FUNCTION_BLOCK "CM_DRVT_N"   // FB148, SCL
{ S7_Optimized_Access := 'FALSE' }
VERSION : 0.0
// --------------------------------------------------------------------------------
//     program     :    CM_DRVT_N
//     description :    calculation of derivative to the order n 
//     name        :    G. Eibelsh鋟ser
//     date        :    31.01.2007
// 
//     revision    :  
//     name        :   
//     date        :    
// 
//                     (c)CGS
//     --------------------------------------------------------------------------------
   VAR_INPUT
      calc_on : Bool;   // calculation activated
      order : Int;   // order of first derivation
      u_in : Real;   // input value
      ts_in : Real;   // sample time
      tc_in : Real;   // call time
      tme_base : Real;
   END_VAR
   VAR_IN_OUT
      y_out : Real;   // output value
   END_VAR
   VAR
      data_rec_init : Bool;   // data record initialisation
      calc_cycle : Int;   // calculation cycle
      i : Int;   // record index
      t : Int;   // time between newest and oldest value in record
      y_t : Real;   // newest value in data record
      y_tn : Real;   // oldest value in data record
      data_rec : Array[0..3600] of Real;   // data record
   END_VAR
BEGIN


       IF #calc_on  THEN        //caculation enabled
           IF #calc_cycle >= REAL_TO_INT(#ts_in / #tc_in)   THEN 
               #calc_cycle  :=  1;

               IF (#order > 3600)   THEN
                   #order   :=  3600;       //limit order to a maximum of 3600
               END_IF;

               IF (#order > 0)  THEN //order of first derivation must be >0

                   //read oldest value from data record
                   //----------------------------------
                   IF (#i = 0) AND #data_rec_init THEN   //record initialisation with new values 
                       #y_tn    :=  #u_in;               //keep y_tn on first input during initialisation
                   ELSIF NOT #data_rec_init THEN 
                       #y_tn    :=  #data_rec[#i];        //write oldest record data to y_tn before overwritting it
                   END_IF;

                   //store new input value in record
                   //-------------------------------
                   #data_rec[#i] :=  #u_in;

                   //read newest value from data record
                   //----------------------------------
                   #y_t :=  #data_rec[#i];

                   //calculation of time between newest and oldest value in record
                   //-------------------------------------------------------------
                   IF #data_rec_init    THEN
                       #t   :=  #i;
                   ELSE
                       #t   :=  #order;
                   END_IF;

                   //calculate first derivation and scale
                   //------------------------------------
                   IF (#t > 0) THEN 
                       #y_out   :=  ((#y_t - #y_tn) / #t) * (#tme_base / #ts_in);
                   END_IF;

                   //increment record index each call
                   //--------------------------------
                   #i   :=  #i + 1;

                   //reset record index when maximum amount of values is reached
                   //-----------------------------------------------------------
                   IF (#i > #order)  THEN
                       #i               :=  0;
                       #data_rec_init   :=  FALSE;
                   END_IF;
               END_IF;
           ELSE   
               #calc_cycle  :=  #calc_cycle + 1;
           END_IF;

       //caculation disabled - reset variables and flags
       //-----------------------------------------------
       ELSE                
           #i               :=  0;
           #y_out           :=  0.0;
           #calc_cycle      :=  1;
           #data_rec_init   :=  TRUE;

       END_IF;
END_FUNCTION_BLOCK

FUNCTION_BLOCK "CM_CALC"   // FB149, SCL
{ S7_Optimized_Access := 'FALSE' }
VERSION : 0.0
// --------------------------------------------------------------------------------
//     program     :    CM_CALC
//     description :    filter calculations 
//     name        :    G. Eibelsh鋟ser
//     date        :    01.07.2020 
// 
//     revision    :    
//     name        :    
//     date        :    
// 
//                     (c)PVA TePla AG
//     --------------------------------------------------------------------------------
   VAR
      S_CAM_1_CTR_X : "CM_PT1";   // PT1
      S_CAM_2_CTR_X : "CM_PT1";   // PT1
      S_CAM_1_RAD_PT : "CM_PT1";   // PT1
      S_CAM_2_RAD_PT : "CM_PT1";   // PT1
      S_CAM_1_DIA_CF : "CM_PT2";   // PT2
      S_CAM_2_DIA_CF : "CM_PT2";   // PT2
      S_CAM_XT_DIA : "CM_PT2";   // PT2
      S_CAM_MLT_LVL_CHG : "CM_PT1";   // PT1
      i : Int;
      scam_mlt_lvl_t1 : Real;
   END_VAR
   VAR CONSTANT
      x_resolution : Real := 2063.0;
      mlt_lvl_chg_rng : Real := 100.0;
   END_VAR
BEGIN

       //stereo camera
       //-------------
       //center x- coordinate of circle fit camera 1
       //-------------------------------------------
       #S_CAM_1_CTR_X  (u_in      := "AV".S_CAM_1_ACT_CF_CTR_X,   //read actual pixel value                  
                       t1_in     := 15.0,                      //delay time T1
                       ts_in     := 0.1,
                       tc_in     := 0.1,
                       range_in  := #x_resolution,
                       range_out := #x_resolution,
                       y_llim    := 0.0,
                       y_hlim    := #x_resolution,
                       y_out     := "AV".S_CAM_1_AVG_CF_CTR_X);  //write average value - not used

       //center x- coordinate of circle fit camera 2
       //-------------------------------------------
       #S_CAM_2_CTR_X  (u_in      := "AV".S_CAM_2_ACT_CF_CTR_X,   //read actual pixel value                    
                       t1_in     := 15.0,                      //delay time T1
                       ts_in     := 0.1,
                       tc_in     := 0.1,
                       range_in  := #x_resolution,
                       range_out := #x_resolution,
                       y_llim    := 0.0,
                       y_hlim    := #x_resolution,
                       y_out     := "AV".S_CAM_2_AVG_CF_CTR_X);  //write average value - not used

       //radius point of camera 1
       //------------------------
       #S_CAM_1_RAD_PT (u_in      := "AV".S_CAM_1_ACT_RAD_PT,     //read actual pixel value                  
                       t1_in     := 15.0,                      //delay time T1
                       ts_in     := 0.1,
                       tc_in     := 0.1,
                       range_in  := #x_resolution,
                       range_out := #x_resolution,
                       y_llim    := 0.0,
                       y_hlim    := #x_resolution,
                       y_out     := "AV".S_CAM_1_AVG_RAD_PT);    //write average value - used for calculation of delta_r and delta_h

       //radius point of camera 2
       //------------------------
       #S_CAM_2_RAD_PT (u_in      := "AV".S_CAM_2_ACT_RAD_PT,     //read actual pixel value                  
                       t1_in     := 15.0,                      //delay time T1
                       ts_in     := 0.1,
                       tc_in     := 0.1,
                       range_in  := #x_resolution,
                       range_out := #x_resolution,
                       y_llim    := 0.0,
                       y_hlim    := #x_resolution,
                       y_out     := "AV".S_CAM_2_AVG_RAD_PT);    //write average value - used for calculation of delta_r and delta_h

       //circle fit camera 1 - PT 2 call
       //-------------------------------
       #S_CAM_1_DIA_CF (u_in      := "AV".S_CAM_1_ACT_DIA_CF,     //read actual pixel value                  
                       t1_in     := "AC".CTL_DIA_TF_1,           //delay time T1 - recipe parameter
                       t2_in     := "AC".CTL_DIA_TF_2,           //delay time T2 - recipe parameter
                       ts_in     := 0.1,
                       tc_in     := 0.1,
                       range_in  := #x_resolution,
                       range_out := #x_resolution,
                       y_llim    := 0.0,
                       y_hlim    := #x_resolution,
                       y_out     := "AV".S_CAM_1_AVG_DIA_CF);    //write average value - not used

       //circle fit camera 2 - PT 2 call
       //-------------------------------
       #S_CAM_2_DIA_CF (u_in      := "AV".S_CAM_2_ACT_DIA_CF,     //read actual pixel value                  
                       t1_in     := "AC".CTL_DIA_TF_1,           //delay time T1 - recipe parameter
                       t2_in     := "AC".CTL_DIA_TF_2,           //delay time T2 - recipe parameter
                       ts_in     := 0.1,
                       tc_in     := 0.1,
                       range_in  := #x_resolution,
                       range_out := #x_resolution,
                       y_llim    := 0.0,
                       y_hlim    := #x_resolution,
                       y_out     := "AV".S_CAM_2_AVG_DIA_CF);    //write average value - not used

       //actual crystal diameter - PT 2 call
       //-----------------------------------
       #S_CAM_XT_DIA   (u_in      := "AV".S_CAM_ACT_XT_DIA,       //read actual mm value                  
                       t1_in     := "AC".CTL_DIA_TF_1,           //delay time T1 - recipe parameter
                       t2_in     := "AC".CTL_DIA_TF_2,           //delay time T2 - recipe parameter
                       ts_in     := 0.1,
                       tc_in     := 0.1,
                       range_in  := "CNF".XT_DIA_RANGE,
                       range_out := "CNF".XT_DIA_RANGE,
                       y_llim    := 0.0,
                       y_hlim    := "CNF".XT_DIA_RANGE,
                       y_out     := "AV".S_CAM_AVG_XT_DIA);      //write average value - used for control loop

       //reset filter time to zero while melt level variable is reseted
       //--------------------------------------------------------------
       IF ("LT".RST_MLT_LVL AND (#i <= 5)) THEN
           #scam_mlt_lvl_t1     :=  0.0;
           #i                   :=  #i + 1;
       ELSE
           #scam_mlt_lvl_t1     :=  "PAR_SUB".SCAM_MLT_LVL_T1;
           "LT".RST_MLT_LVL      :=  FALSE;
           #i                   :=  0;
       END_IF;

       //actual crystal melt level change
       //--------------------------------
       #S_CAM_MLT_LVL_CHG  (u_in      := "AV".S_CAM_ACT_MLT_LVL_CHG,      //read actual mm value                  
                           t1_in     := #scam_mlt_lvl_t1,               //delay time T1
                           ts_in     := 0.1,
                           tc_in     := 0.1,
                           range_in  := #mlt_lvl_chg_rng,
                           range_out := #mlt_lvl_chg_rng,
                           y_llim    := #mlt_lvl_chg_rng * (-1),
                           y_hlim    := #mlt_lvl_chg_rng,
                           y_out     := "AV".S_CAM_AVG_MLT_LVL_CHG);     //write average value - used for control loop

       //write display values
       //--------------------                 
       "DIS".S_CAM_ACT_XT_DIA        :=  "AV".S_CAM_AVG_XT_DIA;     
       "DIS".S_CAM_ACT_MLT_LVL_CHG   :=  "AV".S_CAM_AVG_MLT_LVL_CHG;
       "DIS".S_CAM_1_ACT_RAD_PT      :=  "AV".S_CAM_1_AVG_RAD_PT;
       "DIS".S_CAM_2_ACT_RAD_PT      :=  "AV".S_CAM_2_AVG_RAD_PT;
END_FUNCTION_BLOCK

FUNCTION_BLOCK "CM_DIA_CALC"   // FB150, SCL
{ S7_Optimized_Access := 'FALSE' }
VERSION : 0.0
// --------------------------------------------------------------------------------
//     program     :    CM_DIA_CALC
//     description :    calculation of crystal diameter from measured weight signal 
//     name        :    G. Eibelsh鋟ser
//     date        :    12.02.2008
// 
//                     diameter = 2 * SQRT(weight rate / (position increment * PI * density)
// 
//     revision    :  
//     name        :   
//     date        :    
// 
//                     (c)CGS
//     --------------------------------------------------------------------------------
   VAR_INPUT
      calc_on : Bool;   // calculation activated
      ts_in : Real;   // sample time
      tc_in : Real;   // call time
      u_in : Real;   // input value
      pos_inc : Real;
      pi : Real;
      rho_si_sol : Real;
   END_VAR
   VAR_IN_OUT
      y_out : Real;   // output value
   END_VAR
   VAR
      calc_cycle : Int;   // calculation cycle
   END_VAR
BEGIN


       IF #calc_on  THEN        //caculation enabled
           //do calculation
           //--------------
           IF #calc_cycle >= REAL_TO_INT(#ts_in / #tc_in)   THEN  //check calculation cycle 
               #calc_cycle  :=  1;
               //calculate diameter in mm
               //------------------------
               IF (#u_in > 0.0) AND (#pos_inc > 0.0) THEN 
                   #y_out   :=  2 * SQRT(#u_in / (#pos_inc * #pi * #rho_si_sol));          
               END_IF;
           ELSE   
               #calc_cycle  :=  #calc_cycle + 1; //increment calc cycle variable
           END_IF;

       //caculation disabled - reset output variable
       //-------------------------------------------
       ELSE                
           #calc_cycle      :=  1;
           #y_out           :=  0.0;

       END_IF;
END_FUNCTION_BLOCK

FUNCTION_BLOCK "CM_LOOP_AVG_GAP_OFFS"   // FB151, SCL
{ S7_Optimized_Access := 'FALSE' }
VERSION : 0.0
// --------------------------------------------------------------------------------
//     program     :    CM_LOOP_AVG_GAP_OFFS
//     description :    average gap offset controller
//     name        :    G. Eibelsh鋟ser
//     date        :    27.08.2020
// 
//     revision    :    
//     name        :    
//     date        :    
// 
//                     (c)PVA TePla AG
//     --------------------------------------------------------------------------------
   VAR
      GAP_OFFS : "CM_PT1";   // pt1 filter for average offset speed
      AVG_GAP_OFFS : CONT_C;   // Controller for offset speed of the gap control
      int_hold_req : Bool;   // integral hold action request
      ctrl_calls : Int;   // controller call counter
   END_VAR
   VAR_TEMP
      high_lim_active : Bool;   // high limit of controller output is reached
      low_lim_active : Bool;   // low limit of controller output is reached
      int_action_on : Bool;   // integral action on
      der_action_on : Bool;   // derivative action on
      per_out : Word;   // peripherial controller output variable
      p_part_out : Real;   // proportionality component
      i_part_out : Real;   // integral component
      d_part_out : Real;   // derivative component
      eff_act_val : Real;   // effective process variable
      error_sig : Real;   // control deviation
   END_VAR
   VAR CONSTANT
      nc : Real := 0.0;   // "not connected" input
   END_VAR
BEGIN

       //switch on average gap offset control
       //------------------------------------
       IF ("APC".AUTOMATIC AND "SY".CTL_OFFS_SPEED_ON AND NOT "SY".CTL_HTR_1_SMI) THEN        //offset speed control is triggered by gap control on
           "SY".CTL_AVG_OFFS_ON  :=  TRUE;
       ELSE
           "SY".CTL_AVG_OFFS_ON  :=  FALSE;
       END_IF;    

       //call filter algorithm
       //---------------------                                                  
       #GAP_OFFS(u_in       := "CTL".SET_GAP_CTL_OFFS,                          
               t1_in       := "PAR_MAIN".CTL_AVG_GAP_OFFS_TF, 
               ts_in       := 0.1,
               tc_in       := 0.1,
               range_in    := "CNF".MAX_GAP_OFFS,
               range_out   := "CNF".MAX_GAP_OFFS,
               y_llim      := "CNF".MAX_GAP_OFFS * (-1.0),
               y_hlim      := "CNF".MAX_GAP_OFFS,
               y_out       := "CTL".AVG_GAP_CTL_OFFS); 

       //enable of single controller actions
       //----------------------------------- 
       IF ("AC".CTL_AV_OFFS_TI > 0.0)   THEN         //i- part
           #int_action_on   :=  true;
       ELSE
           #int_action_on   :=  false;
       END_IF;

       IF ("AC".CTL_AV_OFFS_TD > 0.0)   THEN         //d-part
           #der_action_on   :=  true;
       ELSE
           #der_action_on   :=  false;
       END_IF;

       //call average gap offset controller 
       //----------------------------------
       #AVG_GAP_OFFS(COM_RST        :=  "KYD".OFFS_CTRL_RST,                  //restart of controller, resets controller values
                   MAN_ON          :=  NOT "SY".CTL_AVG_OFFS_ON,             //switch controller on/off
                   PVPER_ON        :=  false,                              //activate reading of peripherie value
                   P_SEL           :=  true,                               //proportional action on
                   I_SEL           :=  #int_action_on,                      //integral action on
                   INT_HOLD        :=  #int_hold_req,                       //integral action hold
                   I_ITL_ON        :=  false,                              //initialization of the integral action - set value of I_ITLVAL
                   D_SEL           :=  #der_action_on,                      //derivative action on
                   CYCLE           :=  T#100ms,                            //sample time
                   SP_INT          :=  0.0,                                //internal setpoint
                   PV_IN           :=  "CTL".AVG_GAP_CTL_OFFS * (-1),        //process variable input (input polarity changed to negate the output variable)
                   PV_PER          :=  W#16#0000,                          //process variable peripherial input
                   MAN             :=  0.0,                                //hand value as percentaged input
                   GAIN            :=  "AC".CTL_AV_OFFS_GN,                  //controller gain
                   TI              :=  DINT_TO_TIME(REAL_TO_DINT("AC".CTL_AV_OFFS_TI * 1000.0)),  //integration time
                   TD              :=  DINT_TO_TIME(REAL_TO_DINT("AC".CTL_AV_OFFS_TD * 1000.0)),  //derivative time
                   TM_LAG          :=  DINT_TO_TIME(REAL_TO_DINT("AC".CTL_AV_OFFS_T1 * 1000.0)),  //time lag of the derivative action
                   DEADB_W         :=  0.0,                                //dead band of control deviation
                   LMN_HLM         :=  "CNF".AVG_GAP_OFFS_TMP_RNG,           //upper limit of controller output as percentaged value 
                   LMN_LLM         :=  "CNF".AVG_GAP_OFFS_TMP_RNG * (-1.0),  //lower limit of controller output as percentaged value
                   PV_FAC          :=  1.0,                                //process variable factor (used on peripherial input)
                   PV_OFF          :=  0.0,                                //process variable offset
                   LMN_FAC         :=  1.0,                                //output standardization(percentage to physical value)
                   LMN_OFF         :=  0.0,                                //offset of output value
                   I_ITLVAL        :=  0.0,                                //initialization value of the integral action
                   DISV            :=  0.0);                               //disturbance variable            

               //write output variables of PID controller
               //----------------------------------------
               "CTL".Y_AVG_GAP_OFFS  :=  #AVG_GAP_OFFS.LMN;                   //controller output variable as physical value - scaled as temperature increment

               #per_out         :=  #AVG_GAP_OFFS.LMN_PER;                    //peripherial controller output variable
               #high_lim_active :=  #AVG_GAP_OFFS.QLMN_HLM;                   //high limit of controller output is reached
               #low_lim_active  :=  #AVG_GAP_OFFS.QLMN_LLM;                   //low limit of controller output is reached
               #p_part_out      :=  #AVG_GAP_OFFS.LMN_P;                      //proportionality component
               #i_part_out      :=  #AVG_GAP_OFFS.LMN_I;                      //integral component
               #d_part_out      :=  #AVG_GAP_OFFS.LMN_D;                      //derivative component
               #eff_act_val     :=  #AVG_GAP_OFFS.PV;                         //effective process variable 
               #error_sig       :=  #AVG_GAP_OFFS.ER;                         //control deviation

       //write display values of individual controller parts
       //---------------------------------------------------
       "DIS".AVG_GAP_CONT_P:= #p_part_out;   
       "DIS".AVG_GAP_CONT_D:= #d_part_out;
       "DIS".AVG_GAP_CONT_I:= #i_part_out;

       //write dispaly value of average gap offset controller output - temperature increment
       //-----------------------------------------------------------------------------------
       "DIS".SET_AVG_GAP_OFFS_T_INC  := "CTL".Y_AVG_GAP_OFFS; 

       //evaluate controller output limits
       //---------------------------------
       IF #high_lim_active OR #low_lim_active   THEN                 //check controller limits
           IF (#ctrl_calls > 50) THEN                                   
               IF #high_lim_active AND (#i_part_out > 0.0)   THEN 
                   #int_hold_req    :=  true;                       //set integral action on hold
               ELSIF #low_lim_active AND (#i_part_out < 0.0) THEN 
                   #int_hold_req    :=  true;                       //set integral action on hold
               ELSE 
                   #int_hold_req    :=  false;                      //reset integral action on hold
               END_IF;
           ELSE
               #ctrl_calls  :=  #ctrl_calls + 1;                     //count controller calls
           END_IF;
       ELSE
           #ctrl_calls      :=  0;                                  //reset controller call counts
           #int_hold_req    :=  false;                              //reset integral action hold request
       END_IF;
END_FUNCTION_BLOCK

FUNCTION_BLOCK "CM_AVG_MSR_SEN_POS"   // FB152, SCL
{ S7_Optimized_Access := 'FALSE' }
VERSION : 0.0
// --------------------------------------------------------------------------------
//     program     :    CM_AVG_MSR_SEN_POS
//     description :    filter diameter measurement sensor positions 
//     name        :    G. Eibelsh鋟ser
//     date        :    17.06.2009 
// 
//     revision    :  
//     name        :   
//     date        :    
// 
//                     (c)PVA TePla AG
//     --------------------------------------------------------------------------------
   VAR
      PRD_2_CTR_Y : "CM_PT1";   // PT1
      SLD_AVG_CTR_Y : "CM_SLD_AVG";   // sliding average
   END_VAR
BEGIN

       (*
       PRD_2_CTR_Y    (u_in      := AV.ACT_PRD_2_CTR_Y,        //read actual y-position of sensor                    
                       t1_in     := 60.0,                      //delay time T1
                       ts_in     := 0.1,
                       tc_in     := 0.1,
                       range_in  := 479.0,
                       range_out := 479.0,
                       y_llim    := 0.0,
                       y_hlim    := 479.0,
                       y_out     := AV.AVG_PRD_2_CTR_Y);      //write average y-position of sensor
       *)

       //call calculation of sliding average of product 2 center y-coordinate
       //--------------------------------------------------------------------
       #SLD_AVG_CTR_Y ( calc_on :=  true,                                       //averaging activated
                       ts_in   :=  1.0,                                        //sample time
                       tc_in   :=  0.1,                                        //call time
                       order   :=  60,                                         //order of sliding average
                       u_in    :=  "AV".ACT_PRD_2_CTR_Y,                         //actual value of center y-coordinate
                       y_out   :=  "AV".AVG_PRD_2_CTR_Y);                        //average center y-coordinate as sliding average


       //set display value
       //-----------------
       "DIS".AVG_PRD_2_CTR_Y := "AV".AVG_PRD_2_CTR_Y;
END_FUNCTION_BLOCK

FUNCTION_BLOCK "CM_LOOP_MLT_DRIFT"   // FB153, SCL
{ S7_Optimized_Access := 'FALSE' }
VERSION : 0.0
// --------------------------------------------------------------------------------
//     program     :    CM_LOOP_MLT_DRIFT
//     description :    melt drift control loop 
//     name        :    G. Eibelsh鋟ser
//     date        :    09.02.2010
// 
//     revision    :    
//     name        :    
//     date        :    
// 
//                     (c)PVA TePla AG
//     --------------------------------------------------------------------------------
   VAR
      STD_PID : CONT_C;   // standard Siemens controller algorithm
      DT1 : "CM_DT1";   // dt1 filter
      int_hold_req : Bool;   // integral hold action request
      ctl_mlt_drift_on : Bool;
      cycle : Int;
      count : Int;
      ctrl_calls : Int;   // controller call counter
      i : Int;
      set : Real;   // internal set point
      act : Real;   // internal actual value
      hand : Real;   // internal hand value
      ctl_mlt_drift_tf : Real;
      act_mlt_lvl_lft_rte : Real;
   END_VAR
   VAR_TEMP
      high_lim_active : Bool;   // high limit of controller output is reached
      low_lim_active : Bool;   // low limit of controller output is reached
      int_action_on : Bool;   // integral action on
      der_action_on : Bool;   // derivative action on
      per_out : Word;   // peripherial controller output variable
      p_part_out : Real;   // proportionality component
      i_part_out : Real;   // integral component
      d_part_out : Real;   // derivative component
      eff_act_val : Real;   // effective process variable
      error_sig : Real;   // control deviation
   END_VAR
   VAR CONSTANT
      nc : Real := 0.0;   // "not connected input"
   END_VAR
BEGIN


       //build hand value
       //---------------- 
       #hand := #nc;                    

       //build set point
       //---------------
       #set := 0.0;

       //read actual value        
       //-----------------               
       #act := "AV".ACT_MLT_LVL * (-1);                              

       //reset filter time to zero while melt level variable is reseted
       //--------------------------------------------------------------
       IF ("LT".RST_MLT_LVL AND (#i <= 5)) THEN
           #ctl_mlt_drift_tf    :=  0.0;
           #i                   :=  #i + 1;
       ELSE
           #ctl_mlt_drift_tf    :=  "CNF".CTL_MLT_DRIFT_TF;
           "LT".RST_MLT_LVL      :=  FALSE;
           #i                   :=  0;
       END_IF;

       //call derivative algorithm
       //-------------------------
       #DT1 (u_in       := "AV".ACT_MLT_LVL * 600,                    //build actual value   
            td_in      := 0.10,                                    //mm/min                                
            t1_in      := #ctl_mlt_drift_tf,                        //filter time for derivative calculation                 
            ts_in      := 1.0,
            tc_in      := 0.1,
            range_in   := 479.0,                                   //arbitrary range
            range_out  := 479.0,
            y_llim     := -479.0,
            y_hlim     := 479.0,
            y_out      := #act_mlt_lvl_lft_rte);

       //set alarm message
       //-----------------
       IF "SY".CTL_MLT_DRIFT_ON THEN
           IF (ABS(#act_mlt_lvl_lft_rte) > "CNF".MAX_VALID_DRIFT_RTE) THEN
               "FLT".MLT_LVL_MSR_NOT_VALID  :=  TRUE;
           END_IF;
       END_IF;

       //built controller on flag
       //------------------------
       IF "SY".CTL_MLT_LVL_SMI OR "FLT".MLT_LVL_MSR_NOT_VALID OR NOT "APC".AUTOMATIC  THEN 
           "SY".CTL_MLT_DRIFT_ON := FALSE; 
       ELSIF NOT "SY".CTL_CR_SPD_COF_SMI   THEN 
           "SY".CTL_MLT_DRIFT_ON := "DC".CTL_MLT_DRIFT_ON;         
       ELSE 
           "SY".CTL_MLT_DRIFT_ON := ("SY".CTL_MLT_DRIFT_ON AND NOT "KYD".CTL_MLT_DRIFT_OFF) OR "KYD".CTL_MLT_DRIFT_ON;         
       END_IF;

       //set light variable
       //------------------
       "LT".CTL_MLT_DRIFT_ON := "SY".CTL_MLT_DRIFT_ON;                             

       //switch off pressure controller
       //------------------------------ 
       IF NOT "SY".CTL_MLT_DRIFT_ON  THEN 
           #ctl_mlt_drift_on  :=  false;
       END_IF;

       //enable of single controller actions
       //----------------------------------- 
       IF ("PAR_MAIN".CTL_MLT_DRIFT_TI > 0.0)   THEN         //i- part
           #int_action_on   :=  true;
       ELSE
           #int_action_on   :=  false;
       END_IF;

       IF ("PAR_MAIN".CTL_MLT_DRIFT_TD > 0.0)   THEN         //d-part
           #der_action_on   :=  true;
       ELSE
           #der_action_on   :=  false;
       END_IF;

       //call Standard PID controller 
       //----------------------------
       #STD_PID(COM_RST         :=  "KYD".MLT_DRIFT_CTRL_RST,             //restart of controller, resets controller values
               MAN_ON          :=  NOT #ctl_mlt_drift_on,               //switch controller on/off
               PVPER_ON        :=  false,                              //activate reading of peripherie value
               P_SEL           :=  true,                               //proportional action on
               I_SEL           :=  #int_action_on,                      //integral action on
               INT_HOLD        :=  #int_hold_req,                       //integral action hold
               I_ITL_ON        :=  false,                              //initialization of the integral action - set value of I_ITLVAL
               D_SEL           :=  #der_action_on,                      //derivative action on
               CYCLE           :=  T#100ms,                            //sample time
               SP_INT          :=  #set,                                //internal setpoint
               PV_IN           :=  #act,                                //process variable input
               PV_PER          :=  W#16#0000,                          //process variable peripherial input
               MAN             :=  #hand,                               //hand value as percentaged input
               GAIN            :=  "PAR_MAIN".CTL_MLT_DRIFT_GN,                                        //controller gain
               TI              :=  DINT_TO_TIME(REAL_TO_DINT("PAR_MAIN".CTL_MLT_DRIFT_TI * 1000.0)),   //integration time
               TD              :=  DINT_TO_TIME(REAL_TO_DINT("PAR_MAIN".CTL_MLT_DRIFT_TD * 1000.0)),   //derivative time
               TM_LAG          :=  DINT_TO_TIME(REAL_TO_DINT("PAR_MAIN".CTL_MLT_DRIFT_T1 * 1000.0)),   //time lag of the derivative action
               DEADB_W         :=  0.0,                                            //dead band of control deviation
               LMN_HLM         :=  "PAR_MAIN".LIM_MLT_DRIFT_OFFS / "CNF".CR_SPD_COF_RANGE * 100.0,     //upper limit of controller output as percentaged value 
               LMN_LLM         :=  "PAR_MAIN".LIM_MLT_DRIFT_OFFS / "CNF".CR_SPD_COF_RANGE * (- 100.0), //lower limit of controller output as percentaged value
               PV_FAC          :=  1.0,                            //process variable factor (used on peripherial input)
               PV_OFF          :=  0.0,                            //process variable offset
               LMN_FAC         :=  1.0,                            //output standardization(percentage to physical value)
               LMN_OFF         :=  0.0,                            //offset of output value
               I_ITLVAL        :=  0.0,                            //initialization value of the integral action
               DISV            :=  #nc);                            //disturbance variable

               //write output variables of PID controller
               //----------------------------------------
               "CTL".SET_CR_SPD_COF_OFFS  :=  #STD_PID.LMN / 100.0 * "CNF".CR_SPD_COF_RANGE;  //controller output variable as physical value

               #per_out         :=  #STD_PID.LMN_PER;                    //peripherial controller output variable
               #high_lim_active :=  #STD_PID.QLMN_HLM;                   //high limit of controller output is reached
               #low_lim_active  :=  #STD_PID.QLMN_LLM;                   //low limit of controller output is reached
               #p_part_out      :=  #STD_PID.LMN_P;                      //proportionality component
               #i_part_out      :=  #STD_PID.LMN_I;                      //integral component
               #d_part_out      :=  #STD_PID.LMN_D;                      //derivative component
               #eff_act_val     :=  #STD_PID.PV;                         //effective process variable 
               #error_sig       :=  #STD_PID.ER;                         //control deviation

       //evaluate controller output limits
       //---------------------------------
       IF #high_lim_active XOR #low_lim_active   THEN                //check controller limits
           IF (#ctrl_calls > 50) THEN                                   
               IF #high_lim_active AND (#i_part_out > 0.0)   THEN 
                   #int_hold_req    :=  true;                       //set integral action on hold
               ELSIF #low_lim_active AND (#i_part_out < 0.0) THEN 
                   #int_hold_req    :=  true;                       //set integral action on hold
               ELSE 
                   #int_hold_req    :=  false;                      //reset integral action on hold
               END_IF;
           ELSE
               #ctrl_calls  :=  #ctrl_calls + 1;                     //count controller calls
           END_IF;
       ELSE
           #ctrl_calls      :=  0;                                  //reset controller call counts
           #int_hold_req    :=  false;                              //reset integral action hold request
       END_IF;

       //switch on melt drift controller
       //------------------------------- 
       IF "SY".CTL_MLT_DRIFT_ON    THEN 
           #ctl_mlt_drift_on  :=  true;
       END_IF;

       //write display value
       //-------------------
       "DIS".SET_CR_SPD_COF_OFFS  :=  "CTL".SET_CR_SPD_COF_OFFS;   //write controller offset of crucible speed coeffizient to display value

       //manual reset of unvalid melt level measurements
       //-----------------------------------------------
       IF ("KYD".MLT_DRIFT_CTRL_RST  OR ("APC".STATUS <> "APC".BODY))  THEN
           "FLT".MLT_LVL_MSR_NOT_VALID  :=  FALSE;
       END_IF;
END_FUNCTION_BLOCK

FUNCTION_BLOCK "CM_LOOP_DIA_TMP"   // FB154, SCL
{ S7_Optimized_Access := 'FALSE' }
VERSION : 0.0
// --------------------------------------------------------------------------------
//     program     :    CM_LOOP_DIA_TMP
//     description :    diameter temperature controller (WWX)
//     name        :    G. Eibelsh鋟ser
//     date        :    04.03.213
// 
//     revision    :    
//     name        :    
//     date        :    
// 
//                     (c)PVA TePla AG
//     --------------------------------------------------------------------------------
   VAR
      STD_PID : CONT_C;   // standard Siemens controller algorithm
      int_hold_req : Bool;   // integral hold action request
      ctl_dia_tmp_on : Bool;
      lt_ctl_dia_tmp_on : Bool;
      dia_tmp_ctl_enb : Bool;
      ctrl_calls : Int;   // controller call counter
      set : Real;   // internal set point
      act : Real;   // internal actual value
      hand : Real;   // hand value
   END_VAR
   VAR_TEMP
      high_lim_active : Bool;   // high limit of controller output is reached
      low_lim_active : Bool;   // low limit of controller output is reached
      int_action_on : Bool;   // integral action on
      der_action_on : Bool;   // derivative action on
      per_out : Word;   // peripherial controller output variable
      p_part_out : Real;   // proportionality component
      i_part_out : Real;   // integral component
      d_part_out : Real;   // derivative component
      eff_act_val : Real;   // effective process variable
      error_sig : Real;   // control deviation
   END_VAR
   VAR CONSTANT
      nc_bool : Bool := FALSE;   // "not connected input"
      nc_real : Real := 0.0;   // "not connected input"
   END_VAR
BEGIN


       //read set point and actual value
       //-------------------------------
       #set := "AC".SET_XT_DIA;                           
       #act := "AV".ACT_XT_DIA;                                               

       //built controller enable flag
       //----------------------------
       #dia_tmp_ctl_enb :=      ("APC".STATUS = "APC".BODY)                             //body phase active
                           AND (REAL_TO_INT("PAR_MAIN".BY_LEN_DIA_TMP_CTL_ON) >= 0)  //length for activation >= 0
                           AND ("AV".ACT_XT_LEN >= "PAR_MAIN".BY_LEN_DIA_TMP_CTL_ON);  //body crystal length is equal or greater parameter setting

       //built controller on flag
       //------------------------
       IF "APC".AUTOMATIC AND NOT "SY".CTL_HTR_1_SMI THEN 
           "SY".CTL_DIA_TMP_ON := "DC".CTL_DIA_ON AND #dia_tmp_ctl_enb;  
       ELSE 
           "SY".CTL_DIA_TMP_ON := FALSE; 
       END_IF;

       //set light variable
       //------------------
       #lt_ctl_dia_tmp_on:= "SY".CTL_DIA_TMP_ON;                             

       //change polarity of control values
       //---------------------------------
       #set := #set *(-1);                                                          
       #act := #act *(-1);                                               

       //switch off diameter controller
       //------------------------------ 
       IF NOT "SY".CTL_DIA_TMP_ON    THEN 
           #ctl_dia_tmp_on  :=  false;
       END_IF;

       //enable of single controller actions
       //----------------------------------- 
       IF ("AC".CTL_DIA_TMP_TI > 0.0)   THEN     //i- part
           #int_action_on   :=  true;
       ELSE
           #int_action_on   :=  false;
       END_IF;

       IF ("AC".CTL_DIA_TMP_TD > 0.0)   THEN     //d-part
           #der_action_on   :=  true;
       ELSE
           #der_action_on   :=  false;
       END_IF;

       //call Standard PID controller 
       //----------------------------
       #STD_PID(COM_RST         :=  #nc_bool,                                //restart of controller, resets controller values
               MAN_ON          :=  NOT #ctl_dia_tmp_on,                     //switch controller on/off
               PVPER_ON        :=  false,                                  //activate reading of peripherie value
               P_SEL           :=  true,                                   //proportional action on
               I_SEL           :=  #int_action_on,                          //integral action on
               INT_HOLD        :=  #int_hold_req,                           //integral action hold
               I_ITL_ON        :=  false,                                  //initialization of the integral action - set value of I_ITLVAL
               D_SEL           :=  #der_action_on,                          //derivative action on
               CYCLE           :=  T#100ms,                                //sample time
               SP_INT          :=  #set,                                    //internal setpoint
               PV_IN           :=  #act,                                    //process variable input
               PV_PER          :=  W#16#0000,                              //process variable peripherial input
               MAN             :=  #hand / "CNF".HTR_1_TMP_RANGE_HI * 100.0,  //hand value as percentaged input
               GAIN            :=  "AC".CTL_DIA_TMP_GN,                      //controller gain
               TI              :=  DINT_TO_TIME(REAL_TO_DINT("AC".CTL_DIA_TMP_TI * 1000.0)), //integration time
               TD              :=  DINT_TO_TIME(REAL_TO_DINT("AC".CTL_DIA_TMP_TD * 1000.0)), //derivative time
               TM_LAG          :=  DINT_TO_TIME(REAL_TO_DINT("AC".CTL_DIA_TMP_T1 * 1000.0)), //time lag of the derivative action
               DEADB_W         :=  0.0,                            //dead band of control deviation
               LMN_HLM         :=  100.0,                          //upper limit of controller output as percentaged value 
               LMN_LLM         :=  - 100.0,                        //lower limit of controller output as percentaged value
               PV_FAC          :=  1.0,                            //process variable factor (used on peripherial input)
               PV_OFF          :=  0.0,                            //process variable offset
               LMN_FAC         :=  1.0,                            //output standardization(percentage to physical value)
               LMN_OFF         :=  0.0,                            //offset of output value
               I_ITLVAL        :=  0.0,                            //initialization value of the integral action
               DISV            :=  #nc_real);                       //disturbance variable

               //write output variables of PID controller
               //----------------------------------------
               "CTL".Y_DIA_TMP   :=  #STD_PID.LMN / 100.0 * "CNF".HTR_1_TMP_RANGE_HI; //controller output variable as physical value

               #per_out         :=  #STD_PID.LMN_PER;                        //peripherial controller output variable
               #high_lim_active :=  #STD_PID.QLMN_HLM;                       //high limit of controller output is reached
               #low_lim_active  :=  #STD_PID.QLMN_LLM;                       //low limit of controller output is reached
               #p_part_out      :=  #STD_PID.LMN_P;                          //proportionality component
               #i_part_out      :=  #STD_PID.LMN_I;                          //integral component
               #d_part_out      :=  #STD_PID.LMN_D;                          //derivative component
               #eff_act_val     :=  #STD_PID.PV;                             //effective process variable 
               #error_sig       :=  #STD_PID.ER;                             //control deviation

       //track hand value in body phase
       //------------------------------
       IF ("APC".AUTOMATIC AND ("APC".STATUS = "APC".BODY)) THEN 
           #hand    := "CTL".Y_DIA_TMP;   //when controller is switch off during body phase the temperature increment output stays unchanged
       ELSE 
           #hand    := 0.0;
       END_IF;

       //evaluate controller output limits
       //---------------------------------
       IF #high_lim_active XOR #low_lim_active   THEN                //check controller limits
           IF (#ctrl_calls > 50) THEN                                   
               IF #high_lim_active AND (#i_part_out > 0.0)   THEN 
                   #int_hold_req    :=  true;                       //set integral action on hold
               ELSIF #low_lim_active AND (#i_part_out < 0.0) THEN 
                   #int_hold_req    :=  true;                       //set integral action on hold
               ELSE 
                   #int_hold_req    :=  false;                      //reset integral action on hold
               END_IF;
           ELSE
               #ctrl_calls  :=  #ctrl_calls + 1;                     //count controller calls
           END_IF;
       ELSE
           #ctrl_calls      :=  0;                                  //reset controller call counts
           #int_hold_req    :=  false;                              //reset integral action hold request
       END_IF;

       //switch on diameter controller
       //------------------------------ 
       IF "SY".CTL_DIA_TMP_ON    THEN 
           #ctl_dia_tmp_on  :=  true;
       END_IF;

       //controller outputs written to display variables of test controller (temporary 18.07.2013, ge)
       //---------------------------------------------------------------------------------------------
       IF NOT "LT".TEST_CTRL_ON THEN 
           "DIS".TEST_P_PART_OUT :=  #STD_PID.LMN_P;
           "DIS".TEST_I_PART_OUT :=  #STD_PID.LMN_I;
           "DIS".TEST_D_PART_OUT :=  #STD_PID.LMN_D;
           "DIS".TEST_CTRL_OUT   :=  "CTL".Y_DIA_TMP;
       END_IF;
END_FUNCTION_BLOCK

FUNCTION_BLOCK "AM_CTRL"   // FB193, SCL
{ S7_Optimized_Access := 'FALSE' }
VERSION : 0.0
// --------------------------------------------------------------------------------
//     program     :    AM_CTRL
//     description :    apc control module  
//     name        :    K. Kalkowski
//     date        :    01.09.99
// 
//     revision    :    
//     name        :    
//     date        :    
//                     (c)PVA TePla AG
//     --------------------------------------------------------------------------------
   VAR
      emg_sep_start : Bool;   // start flag for emergency separation
      lt_htr_1_on_old : Bool;
      status_old : Int;
      state_prv : Int;
      emg_sep_dly : Int;   // delay time emergency separation mode
      xt_pos_at_start : Real;
      gas_csp_inc : Real;
      pwr_csp_inc : Real;
   END_VAR
   VAR_TEMP
      act_smi_sta : Int;
      dummy_out_real : Real;
      sign : Real;
      status : Real;
      step_no : Real;
   END_VAR
BEGIN


       // set phase number
       // ----------------
       "APC".IDLE         := 0;            //APC # of idle mode
       "APC".CHARGING     := 1;            //APC # of charging mode
       "APC".PUMP_DOWN    := 2;            //APC # of pump down mode
       "APC".MELTING      := 3;            //APC # of melting mode
       "APC".DIPPING      := 4;            //APC # of dipping mode
       "APC".NECK         := 5;            //APC # of neck mode
       "APC".SHOULDER     := 6;            //APC # of shoulder mode
       "APC".BODY         := 7;            //APC # of body mode
       "APC".ENDCONE      := 8;            //APC # of endcone mode
       "APC".SHUT_DOWN    := 9 ;           //APC # of shut down mode
       "APC".REMOVAL      := 10;           //APC # of removal mode
       "APC".EMG          := 11;           //APC # of emergency separation mode

       //set state numbers
       //-----------------
       "APC".STATE_STD_BY        := 1;   //APC # of state standby
       "APC".STATE_SERV          := 2;   //APC # of state service
       "APC".STATE_RUN           := 3;   //APC # of state process run
       "APC".STATE_VAC_TEST      := 4;   //APC # of state vacuum test without melting
       "APC".STATE_LOADING       := 5;   //APC # of state loading
       "APC".STATE_MAINTENANCE   := 6;   //APC # of state maintenance
       "APC".STATE_ENGINEERING   := 7;   //APC # of state engineering
       "APC".STATE_BAKE_OUT      := 8;   //APC # of state bake out

       //set machine state
       //-----------------
       IF "KYD".STATE_STD_BY THEN 
           "STA".ACT_STATE   :=  "APC".STATE_STD_BY;
       ELSIF "KYD".STATE_SERV    THEN
           "STA".ACT_STATE   :=  "APC".STATE_SERV;
       ELSIF "KYD".STATE_RUN THEN
           "STA".ACT_STATE   :=  "APC".STATE_RUN;
       ELSIF "KYD".STATE_VAC_TEST THEN
           "STA".ACT_STATE   :=  "APC".STATE_VAC_TEST;
       ELSIF "KYD".STATE_LOADING THEN
           "STA".ACT_STATE   :=  "APC".STATE_LOADING;
       ELSIF "KYD".STATE_MAINTENANCE THEN
           "STA".ACT_STATE   :=  "APC".STATE_MAINTENANCE;
       ELSIF "KYD".STATE_ENGINEERING THEN
           "STA".ACT_STATE   :=  "APC".STATE_ENGINEERING;
       ELSIF "KYD".STATE_BAKE_OUT THEN
           "STA".ACT_STATE   :=  "APC".STATE_BAKE_OUT;
       END_IF;

       //detect end of process run, vacuum test and bake out
       //---------------------------------------------------
       IF ("STA".ACT_STATE = "APC".STATE_RUN) OR 
           ("STA".ACT_STATE = "APC".STATE_VAC_TEST) OR 
           ("STA".ACT_STATE = "APC".STATE_BAKE_OUT)        THEN     //run, vacuum test or bake out state is active

           IF ((#status_old <> "APC".IDLE) AND ("APC".STATUS = "APC".IDLE)) THEN  //phase switched from "not IDLE" to "IDLE"
               "STA".ACT_STATE   :=  "APC".STATE_SERV;         //activate state "setup"
           END_IF;
       //detect end of loading
       //---------------------
       ELSIF ("STA".ACT_STATE = "APC".STATE_LOADING) THEN
           IF ("LT".ENB_LOADING AND "KYD".LOADING_DONE) THEN   //loading is enabled and loading done acknowledged
               "STA".ACT_STATE   :=  "APC".STATE_SERV;
           END_IF;
       END_IF;

       #status_old  :=  "APC".STATUS; //store last actual status

       //calculation of total gas and power consumption of process run
       //-------------------------------------------------------------
       IF (("STA".ACT_STATE = "APC".STATE_RUN) AND (#state_prv <> "APC".STATE_RUN)) THEN  //detect start of process run
           "AV".TOT_GAS_CSP  :=  0.0;                                                //reset total gas consumption
           "AV".TOT_PWR_CSP  :=  0.0;                                                //reset total power consumption
           #gas_csp_inc     :=  0.0;                                                //reset gas consumption increment
           #pwr_csp_inc     :=  0.0;                                                //reset power consumption increment
       ELSIF ("STA".ACT_STATE = "APC".STATE_RUN) THEN
           IF "SysTick100ms" THEN                                                    //calculate every 100ms
               //calcualate gas consumption increments in 100ms interval
               //-------------------------------------------------------
               IF ("LT".V5_OPEN OR "LT".V6_OPEN) THEN          //inlet valve is open
                   #gas_csp_inc :=  #gas_csp_inc + "P_BM_ACT_GAS_FLW_MFC_1":P / 600.0;
               END_IF;
               //calcualate power consumption increments in 100ms interval
               //---------------------------------------------------------
               IF ("LT".HTR_1_ON OR "LT".HTR_2_ON) THEN        //heater is on  
                   #pwr_csp_inc     :=  #pwr_csp_inc + ("AV".ACT_HTR_1_PWR + "AV".ACT_HTR_2_PWR) / 36000.0;
               END_IF;
           END_IF;

           //total gas consumption in [l]
           //----------------------------
           IF (#gas_csp_inc >= 0.1) THEN 
               "AV".TOT_GAS_CSP  :=  "AV".TOT_GAS_CSP + #gas_csp_inc;   //total gas consumption in [l] - only inlet V5 and V6 (MFC)   
               #gas_csp_inc     :=  0.0;
           END_IF;

           //total power consumption in [KWh]
           //-------------------------------
           IF (#pwr_csp_inc >= 0.1) THEN 
               "AV".TOT_PWR_CSP  :=  "AV".TOT_PWR_CSP + #pwr_csp_inc;   
               #pwr_csp_inc     :=  0.0;
           END_IF;
       END_IF;

       #state_prv   := "STA".ACT_STATE;   //store last actual state

       //display total gas and power consumption
       //---------------------------------------
       "DIS".TOT_GAS_CSP  :=  "AV".TOT_GAS_CSP;
       "DIS".TOT_PWR_CSP  :=  "AV".TOT_PWR_CSP;

       //monitor melt temperature in melting phase
       //-----------------------------------------
       IF  ("APC".STATUS = "APC".MELTING)                      AND
           ("PAR_MAIN".ME_MAX_MLT_TMP >= 900.1)              AND
           ("CTL".AVG_MLT_1_TMP > "PAR_MAIN".ME_MAX_MLT_TMP)   THEN

           "FLT".ME_MLT_TMP_TOO_HI   :=  TRUE;
       ELSE
           "FLT".ME_MLT_TMP_TOO_HI   :=  FALSE;
       END_IF;

       //reset automatic operator call
       //-----------------------------
       IF "KYD".ACKN_AUTO_OP_CALL THEN
           "LT".AUTO_OP_CALL   :=  FALSE;
       END_IF;

       //built automatic operator call flag
       //----------------------------------
       IF "LT".AUTO_OP_CALL THEN 
           IF "SysTick2s" AND NOT "DV".AUTO_OP_CALL THEN
               "DV".AUTO_OP_CALL := TRUE;                                        //call flag on 2s cycle
           ELSIF  "SysTick200ms" AND "DV".AUTO_OP_CALL THEN
               "DV".AUTO_OP_CALL := FALSE;
           END_IF;
       ELSE       
           "DV".AUTO_OP_CALL := FALSE;
       END_IF;       

       // calculate total length
       // ----------------------
       IF (("APC".STATUS >= "APC".PUMP_DOWN) AND ("APC".STATUS <= "APC".DIPPING))   THEN
           "AV".ACT_TOT_XT_LGH  :=  0.0;
       //neck restart
       //-----------
       ELSIF "DV".NE_RESTART THEN            //set in FB AM_NE step 200
           #xt_pos_at_start     :=  "AV".ACT_XT_POS;
           "AV".ACT_TOT_XT_LGH   :=  0.0;
           "DV".NE_RESTART       :=  FALSE;
       //crystal growth
       //--------------
       ELSIF (("APC".STATUS >= "APC".NECK) AND ("APC".STATUS <= "APC".ENDCONE))   THEN 
           //gap control activated
           //---------------------
           IF (("CNF".ACT_DVC_CNF AND 2#0100_0000_0000_0000_0000_0000_0000_0000) = 2#0100_0000_0000_0000_0000_0000_0000_0000) THEN
                   // Calculate total crystal length from crystal lift speed set point
                   //-----------------------------------------------------------------
                   IF "SysTick100ms" THEN
                       "AV".ACT_TOT_XT_LGH:= "AV".ACT_TOT_XT_LGH + ("CTL".SET_XT_SPD * 1/600.0);

                   END_IF;
           //no gap control activated
           //------------------------
           ELSE 
               //call total length calculation
               //-----------------------------
               "AM_CALC_LENGTH" (start_pos       := #xt_pos_at_start,
                               actual_pos      := "AV".ACT_XT_POS,
                               total_len       := -1.0,              // % not calculated
                               actual_len      => "AV".ACT_TOT_XT_LGH,
                               actual_len_prc  => #dummy_out_real);
           END_IF; 
       END_IF;

       "DIS".ACT_TOT_XT_LGH  :=  "AV".ACT_TOT_XT_LGH;

       // weight of remaining Si charge (liquid) in crucible
       // --------------------------------------------------
       "CRUC".ACT_CR_WGT := "PAR_MAIN".CH_SILICON_CHARGE
                              - "CRUC".ACT_XT_WGT_SUM            //calculated in FC CM_CALC_NEXT_BY
                              - "AV".ACT_XT_WGT_CALC;            //calculated in ekz_bm_weight_calc with rho_si_sol

       // show remaining Si charge in crucible
       // ------------------------------------ 
       "DIS".ACT_SI_CRG_WGT := "CRUC".ACT_CR_WGT;

       // set operating mode
       // ------------------
       "APC".AUTOMATIC   :=          "PDI".EMO             
                           AND     "DC".MOD_AUT_ENB   
                           AND NOT "KYD".MOD_MANUAL 
                           AND     ("KYD".MOD_AUTO OR "APC".AUTOMATIC);

       "LT".MOD_AUTO     :=  "APC".AUTOMATIC;
       "LT".MOD_MANUAL   :=  NOT "APC".AUTOMATIC;
       "APC".CONT        :=  "KYD".MOD_CONTINUE;

       //set light variable for displaying remaining melt value
       //------------------------------------------------------
       IF "DV".NEW_SI_CRG_WGT_CALC   THEN
           "LT".SI_CRG_WGT_VALID     :=  TRUE;
           "DV".NEW_SI_CRG_WGT_CALC  :=  FALSE;
       END_IF;

       //reset light variable for displaying remaining melt value
       //--------------------------------------------------------
       IF  ("APC".STATUS = "APC".ENDCONE)      OR                  //endcone or pump down phase
           ("APC".STATUS = "APC".PUMP_DOWN)    THEN  

           "LT".SI_CRG_WGT_VALID :=  FALSE;

       ELSIF ("APC".STATUS >= "APC".NECK) AND ("APC".STATUS <= "APC".BODY) THEN        //neck, shoulder and body phase
           IF "LT".XT_LFT_DN THEN                                                //xtal down, remelting
               "LT".SI_CRG_WGT_VALID :=  FALSE;
           END_IF;
       END_IF;

       //disable showing of target temperature set point outside removal phase
       //---------------------------------------------------------------------
       IF (("APC".STATUS <> "APC".REMOVAL) OR ("DIS".RE_HTR_1_TRG_SET_TMP <= "AC".SET_HTR_1_TMP)) THEN
           "LT".SHOW_HTR_1_TRG_TMP   :=  FALSE;
       END_IF;

       //set crystal removed flag
       //------------------------
       IF ("APC".STATUS = "APC".REMOVAL) AND "LT".SHOW_XT_RMV_BTN THEN
           IF "KYD".RE_XT_RMV THEN
               "DV".MAN_ACKN_XT_RMV  :=  TRUE;
           END_IF;
       ELSE
           "DV".MAN_ACKN_XT_RMV  :=  FALSE;
       END_IF;

       //call semi automatic function
       //----------------------------
       "AM_SEMI_AUTO"();

       //call crucible position monitoring
       //---------------------------------
       "CM_CR_POS_MON"();

       //display crystal length
       //----------------------
       "DIS".ACT_XT_LEN_MM   :="AV".ACT_XT_LEN;
       "DIS".ACT_XT_LEN_PERC :="AV".ACT_XT_LEN_PRC;

       // show actual process status
       // --------------------------
       "STA".ACT_PROCESS  := "APC".STATUS;       
       "STA".ACT_OP_MSG   := "APC".OP_MSG;
       "STA".ACT_TME_TOT  := "APC".ACT_TME_TOT;          // total time
       "STA".ACT_TME_PROC := "APC".ACT_TME_PROC;         // process time (for each phase)

       IF ("APC".ACT_TME_STE < 0) THEN
           "STA".ACT_TME_STE  := 0;
       ELSE
           "STA".ACT_TME_STE  := "APC".ACT_TME_STE;      // step time (till end of step)
       END_IF;

       IF ("APC".STATUS = "APC".IDLE) THEN
           "STA".ACT_STE_NO := "AM_ID_DB".active_step[0];   // for debuging only
       END_IF;
       IF ("APC".STATUS = "APC".PUMP_DOWN) THEN
           "STA".ACT_STE_NO := "AM_PD_DB".active_step[0];   // for debuging only
       END_IF;
       IF ("APC".STATUS = "APC".MELTING) THEN
           "STA".ACT_STE_NO := "AM_ME_DB".active_step[0];   // for debuging only
       END_IF;
       IF ("APC".STATUS = "APC".DIPPING) THEN
           "STA".ACT_STE_NO := "AM_DI_DB".active_step[0];   // for debuging only
       END_IF;
       IF ("APC".STATUS = "APC".NECK) THEN
           "STA".ACT_STE_NO := "AM_NE_DB".active_step[0];   // for debuging only
       END_IF;
       IF ("APC".STATUS = "APC".SHOULDER) THEN
           "STA".ACT_STE_NO := "AM_SH_DB".active_step[0];   // for debuging only
       END_IF;
       IF ("APC".STATUS = "APC".BODY) THEN
           "STA".ACT_STE_NO := "AM_BY_DB".active_step[0];   // for debuging only
       END_IF;
       IF ("APC".STATUS = "APC".ENDCONE) THEN
           "STA".ACT_STE_NO := "AM_EC_DB".active_step[0];   // for debuging only
       END_IF;
       IF ("APC".STATUS = "APC".SHUT_DOWN) THEN
           "STA".ACT_STE_NO := "AM_SD_DB".active_step[0];   // for debuging only
       END_IF;
       IF ("APC".STATUS = "APC".REMOVAL) THEN
           "STA".ACT_STE_NO := "AM_RE_DB".active_step[0];   // for debuging only
       END_IF;
       IF ("APC".STATUS = "APC".EMG) THEN
           "STA".ACT_STE_NO := "AM_EMG_DB".active_step[0];   // for debuging only
       END_IF;

       // set request from PC
       // -------------------
       IF NOT ("DV".EMG_DRV_ENB OR "LT".EMG_MOD_REQ)    THEN    // emergency mode deactivated ?

           IF ("KYD".MOD_STOP) THEN 
               "APC".REQUEST := 0;
           END_IF;

           IF ("KYD".MOD_START) THEN 
               "APC".REQUEST := 2;
               "APC".PD_WITH_ME := TRUE;
           END_IF;

           IF ("KYD".MOD_PUMP_DOWN) THEN 
               "APC".REQUEST := 2;
               "APC".PD_WITH_ME := FALSE;
           END_IF;

           IF ("KYD".MOD_MELTING) THEN 
               "APC".REQUEST := 3;
           END_IF;

           IF ("STA".ACT_STATE <> "APC".STATE_BAKE_OUT) THEN   //all machine states except bake out
               IF ("KYD".MOD_DIP) THEN 
                   "APC".REQUEST                 := 4;
                   "APC".MOVE_CRUC_INTO_DIP_POS  := "KYD".MOVE_CR_FOR_DIP;
                   "KYD".MOVE_CR_FOR_DIP         := FALSE;
                   "APC".BYRST                   := FALSE;
                   "APC".CALC_LEN2               := FALSE;
               END_IF;
               IF ("KYD".DIP2) THEN 
                   "APC".REQUEST                 := 4;
                   "APC".MOVE_CRUC_INTO_DIP_POS  := "KYD".MOVE_CR_FOR_DIP;
                   "KYD".MOVE_CR_FOR_DIP         := FALSE;
                   "APC".BYRST                   := TRUE;
                   "APC".CALC_LEN2               := FALSE;
               END_IF;
               IF ("KYD".DIP2_NEW_LEN) THEN 
                   "APC".REQUEST                 := 4;
                   "APC".MOVE_CRUC_INTO_DIP_POS  := "KYD".MOVE_CR_FOR_DIP;
                   "KYD".MOVE_CR_FOR_DIP         := FALSE;
                   "APC".BYRST                   := TRUE;
                   "APC".CALC_LEN2               := TRUE;
               END_IF;

               IF ("KYD".MOD_NECK) THEN 
                   "APC".REQUEST := 5;
               END_IF;

               IF ("KYD".MOD_SHOULDER) THEN 
                   "APC".REQUEST := 6;
               END_IF;

               IF ("KYD".MOD_BODY) THEN 
                   "APC".REQUEST := 7;
               END_IF;

               IF ("KYD".MOD_ENDCONE) THEN 
                   "APC".REQUEST := 8;
                   "APC".SUTDN   := TRUE;
                   "APC".PNBDY   := FALSE;
               END_IF;
               IF ("KYD".ENDCONE_NO_SD) THEN 
                   "APC".REQUEST := 8;
                   "APC".SUTDN   := FALSE;
                   IF ("APC".STATUS = "APC".BODY) THEN
                       "APC".PNBDY   := TRUE;        // 2nd body if body and no shut down
                   ELSE
                       "APC".PNBDY   := FALSE;
                   END_IF;
               END_IF;

               IF ("KYD".MOD_REMOVAL) THEN     
                   "APC".REQUEST := 10;
                   IF ("APC".STATUS = "APC".BODY) THEN
                       "APC".RE_WHILE_BY := TRUE;        // removal started during body mode
                   ELSE
                       "APC".RE_WHILE_BY := FALSE;
                   END_IF;
               END_IF;
           END_IF;

           IF ("KYD".MOD_SHUT_DOWN) THEN 
               "APC".REQUEST := 9;
           END_IF;

       END_IF;

       //start emergency phase
       //---------------------
       IF ("APC".STATUS = "APC".NECK)         OR 
           ("APC".STATUS = "APC".SHOULDER)    OR
           ("APC".STATUS = "APC".BODY)        OR
           ("APC".STATUS = "APC".ENDCONE)     THEN

           IF (#lt_htr_1_on_old <> "LT".HTR_1_ON) AND ("LT".HTR_1_ON = false) THEN //detect change from heater on to heater off 
            "DV".HOR_OPP    := TRUE;
            "DV".LMP_OR     := TRUE;
            "LT".EMG_MOD_REQ := TRUE;        //show window with cancel button on PC
           END_IF;

           #lt_htr_1_on_old := "LT".HTR_1_ON;        

           IF ("KYD".MOD_EMG_OFF OR "LT".HTR_1_ON) THEN
            "DV".HOR_OPP    := FALSE;
            "DV".LMP_OR     := FALSE;
            "LT".EMG_MOD_REQ := FALSE;
           END_IF;

            #emg_sep_start    := "SysOndelay"(DIN := "LT".EMG_MOD_REQ,
                                           SetTime := REAL_TO_INT("PAR_MAIN".MCONST_EMG_WAIT_TME), 
                                           Tick := "SysTick1s",
                                           ActTime := #emg_sep_dly );

            IF "LT".EMG_MOD_REQ THEN                 //calculate time till emergency separation is started
                "DIS".ACT_TME_TILL_EMG := "PAR_MAIN".MCONST_EMG_WAIT_TME - #emg_sep_dly;
               IF "DIS".ACT_TME_TILL_EMG < 0.0 THEN
                   "DIS".ACT_TME_TILL_EMG := 0.0;
               END_IF;
            ELSE
               "DIS".ACT_TME_TILL_EMG := 0.0;
            END_IF;

            IF #emg_sep_start THEN
               "LT".EMG_MOD_REQ  := false;    
               "APC".REQUEST     :=  11;
            END_IF;


       END_IF;    

       // reset keys
       // ----------
       "KYD".MOD_STOP := FALSE;
       "KYD".MOD_START := FALSE;
       "KYD".MOD_PUMP_DOWN := FALSE;
       "KYD".MOD_MELTING := FALSE;
       "KYD".MOD_DIP := FALSE;
       "KYD".MOD_NECK := FALSE;
       "KYD".MOD_SHOULDER := FALSE;
       "KYD".MOD_BODY := FALSE;
       "KYD".MOD_ENDCONE := FALSE;
       "KYD".MOD_SHUT_DOWN := FALSE;
       "KYD".MOD_REMOVAL := FALSE;
       "KYD".MOD_CONTINUE := FALSE;
       "KYD".DIP2 := FALSE;             
       "KYD".DIP2_NEW_LEN := FALSE;
       "KYD".ENDCONE_NO_SD := FALSE;
       // KYD.MOVE_CR_FOR_DIP := FALSE;    this flag is reset above 


       // set request from apc
       // --------------------
       IF ("DC".MOD_ID) THEN "APC".REQUEST := 0;
       END_IF;
       IF ("DC".MOD_PD) THEN "APC".REQUEST := 2;
           "APC".PD_WITH_ME := TRUE;
       END_IF;
       IF ("DC".MOD_ME) THEN "APC".REQUEST := 3;
       END_IF;
       IF ("DC".MOD_DI) THEN "APC".REQUEST := 4;
       END_IF;
       IF ("DC".MOD_NE) THEN "APC".REQUEST := 5;
       END_IF;
       IF ("DC".MOD_SH) THEN "APC".REQUEST := 6;
       END_IF;
       IF ("DC".MOD_BY) THEN "APC".REQUEST := 7;
       END_IF;
       IF ("DC".MOD_EC) THEN "APC".REQUEST := 8;
       END_IF;
       IF ("DC".MOD_SD) THEN "APC".REQUEST := 9;
       END_IF;
       IF ("DC".MOD_RE) THEN "APC".REQUEST := 10;
       END_IF;

       // reset flags
       // -----------
       "DC".MOD_ID := FALSE;
       "DC".MOD_PD := FALSE;
       "DC".MOD_ME := FALSE;
       "DC".MOD_DI := FALSE;
       "DC".MOD_NE := FALSE;
       "DC".MOD_SH := FALSE;
       "DC".MOD_BY := FALSE;
       "DC".MOD_EC := FALSE;
       "DC".MOD_SD := FALSE;
       "DC".MOD_RE := FALSE;


       // start sequence
       // --------------
       IF "APC".REQUEST <> 99 THEN
           CASE "APC".REQUEST OF                                     //start process mode
               0    :                                                  //start idle mode      
                   "AM_ID_DB"(start     := true);
               1    :                                                  //start charging mode
                   "AM_PD_DB"(start     := true);
               2    :                                                  //start pump down mode
                   "AM_PD_DB"(start     := true);
               3    :                                                  //start melting mode
                   "AM_ME_DB"(start     := true);
               4    :                                                  //start dipping mode
                   "AM_DI_DB"(start     := true);
               5    :                                                  //start neck mode
                   "AM_NE_DB"(start     := true);
               6    :                                                  //start shoulder mode
                   "AM_SH_DB"(start     := true);
               7    :                                                  //start body mode
                   "AM_BY_DB"(start     := true);
               8    :                                                  //start end cone mode
                   "AM_EC_DB"(start     := true);
               9    :                                                  //start shut down mode  
                   "AM_SD_DB"(start     := true);
               10   :                                                  //start removal mode
                   "AM_RE_DB"(start     := true);
               11   :                                                  //start emergency separation mode
                   "AM_EMG_DB"(start     := true);

               ELSE :                                                  //apc request error
               // error code:  apc request error
               ;
           END_CASE;
           "APC".REQUEST := 99;    
       END_IF;


       // do automatic sequence
       // ---------------------
       CASE "APC".STATUS OF                                         //do process mode
           0    :                                                      //do idle
               "AM_ID_DB"(start    := false);
           1    :                                                      //do charging
               "AM_PD_DB"(start    := false);
           2    :                                                      //do pump down
               "AM_PD_DB"(start    := false);
           3    :                                                      //do melting
               "AM_ME_DB"(start    := false);
           4    :                                                      //do dipping
               "AM_DI_DB"(start    := false);
           5    :                                                      //do neck
               "AM_NE_DB"(start    := false);
           6    :                                                      //do shoulder
               "AM_SH_DB"(start    := false);
           7    :                                                      //do body
               "AM_BY_DB"(start    := false);
           8    :                                                      //do end cone
               "AM_EC_DB"(start    := false);
           9    :                                                      //do shut down
               "AM_SD_DB"(start    := false);
           10    :                                                     //do removal
               "AM_RE_DB"(start    := false);
           11    :                                                     //do emergency separation
               "AM_EMG_DB"(start  := false);


       END_CASE;

       // show active status
       // ------------------
       "LT".MOD_STOP      := ("APC".STATUS = 0);
       "LT".MOD_PUMP_DOWN := ("APC".STATUS = 2);
       "LT".MOD_MELTING   := ("APC".STATUS = 3);
       "LT".MOD_DIP       := ("APC".STATUS = 4);
       "LT".MOD_NECK      := ("APC".STATUS = 5);
       "LT".MOD_SHOULDER  := ("APC".STATUS = 6);
       "LT".MOD_BODY      := ("APC".STATUS = 7);
       "LT".MOD_ENDCONE   := ("APC".STATUS = 8);
       "LT".MOD_SHUT_DOWN := ("APC".STATUS = 9);
       "LT".MOD_REMOVAL   := ("APC".STATUS = 10);
       "LT".MOD_EMG       := ("APC".STATUS = 11);

       "LT".PMELT         := "APC".PD_WITH_ME;        // pump down with melting
       "LT".PNBDY         := "APC".PNBDY;             // data for 1st body saved
       "LT".BYRST         := "APC".BYRST;             // 2nd body started
       "LT".SUTDN         := "APC".SUTDN;             // endcone with shut down
       "LT".LEN2_CALC     := "APC".LEN2_CALC;         // length for 2nd body calculated


       //evaluation of phase status and semi automatic
       //---------------------------------------------
       IF "APC".AUTOMATIC    THEN    //set sign variable according operation mode
           #sign    :=  1.0;         //automatic mode
       ELSE
           #sign    :=  - 1.0;       //manual mode
       END_IF;

       //convert status and step number variables
       //----------------------------------------
       #status  :=  INT_TO_REAL("APC".STATUS);
       #step_no :=  INT_TO_REAL("STA".ACT_STE_NO);

       //calculate display value phase status
       //------------------------------------
       "DIS".ACT_PHA_STA :=  (#status + #step_no / 10000.0) * #sign;


       //calculate actual semi automatic status
       //--------------------------------------
       #act_smi_sta :=  0;                          //init status variable

       IF "SY".CTL_DIA_SMI   THEN                    //crystal speed  
           #act_smi_sta :=  #act_smi_sta + 1;
       END_IF;
       IF "SY".CTL_XT_ROT_SMI    THEN                //crystal rotation
           #act_smi_sta :=  #act_smi_sta + 2;
       END_IF;
       IF "SY".CTL_MLT_LVL_SMI   THEN
           #act_smi_sta :=  #act_smi_sta + 4;        //crucible speed
       END_IF;    
       IF "SY".CTL_CR_ROT_SMI    THEN
           #act_smi_sta :=  #act_smi_sta + 8;        //crucible rotation
       END_IF;
       IF "SY".CTL_HTR_1_SMI    THEN                  
           #act_smi_sta :=  #act_smi_sta + 16;       //heater 1
       END_IF;
       IF "SY".CTL_HTR_2_SMI    THEN                 
           #act_smi_sta :=  #act_smi_sta + 32;       //heater 2 power
       END_IF;
       IF "SY".CTL_GAS_FLOW_SMI    THEN              
           #act_smi_sta :=  #act_smi_sta + 64;       //gas flow
       END_IF;
       IF "SY".CTL_PRS_SMI    THEN                   
           #act_smi_sta :=  #act_smi_sta + 128;      //pressure
       END_IF;
       IF "SY".CTL_MAG_1_SMI    THEN                 
           #act_smi_sta :=  #act_smi_sta + 256;      //magnet current
       END_IF;
       IF "SY".CTL_CR_SPD_COF_SMI   THEN
           #act_smi_sta :=  #act_smi_sta + 512;      //crucible speed coeffizient
       END_IF;
       IF "SY".CTL_GAP_SMI THEN
           #act_smi_sta :=  #act_smi_sta + 1024;     //gap control
       END_IF;

       //write display value of semi automatic status
       //--------------------------------------------   
       "DIS".ACT_SMI_STA :=  #act_smi_sta;
END_FUNCTION_BLOCK

FUNCTION_BLOCK "AM_ID"   // FB195, SCL
{ S7_Optimized_Access := 'FALSE' }
VERSION : 0.0
// --------------------------------------------------------------------------------
//     program     :    AM_ID
//     description :    apc idle module  
//     name        :    D. Bruess
//     date        :    24.08.99
// 
//     revision    :    
//     name        :    
//     date        :    
//                     (c)CGS
//     --------------------------------------------------------------------------------
   VAR_INPUT
      start : Bool;   // start sequence, activate step 10 (impulse triggered)
   END_VAR
   VAR
      start_previous : Bool;   // start input value of last call
      cont_previous : Bool;   // cont input value of last call
      resume_previous : Bool;   // resume input value of last call
      jump_previous : Bool;   // jump input value of last call
      single_previous : Bool;   // single input value of last call
      active_step : Array[0..7] of Int;   // active step number for sequence level 0..7
      next_step : Array[0..7] of Int;   // next step number for sequence level 0..7
      hold_step : Array[0..7] of Int;   // step number of step on hold
      end_of_step : Array[0..7] of Bool;   // active step is done flag for sequence 0..7
      EndOfStep : Bool;   // default value for active step is done flag
      cont_enable : Array[0..7] of Bool;   // enable continue function
      ContEnable : Bool;   // default value for enable continue function
   END_VAR
BEGIN


       "APC".STATUS := "APC".IDLE;                                     // set apc status               

       "AM_SEQUENCE_CTL" (start_p            := #start,               // control sequence
                        start_previous_p   := #start_previous,
                        cont_previous_p    := #cont_previous, 
                        resume_previous_p  := #resume_previous,
                        jump_previous_p    := #jump_previous,
                        single_previous_p  := #single_previous,
                        active_step_p      := #active_step, 
                        next_step_p        := #next_step,
                        hold_step_p        := #hold_step, 
                        end_of_step_p      := #end_of_step, 
                        cont_enable_p      := #cont_enable); 



       CASE #active_step[0] OF    //sequence level_0
   //step--0-----level--0-------------------------------------------------off--(sequence off)--------------
           0    :                                                  
                #next_step[0] := 0;

   //step--1-----level--0-------------------------------------------------hold-(test sequence)-------------
           1   :                                                       
               IF #next_step[0] = #active_step[0] THEN                   //init step     
                   //init code
                   ; 
               END_IF;

               //step code                                             //do step
               ;

   //-step-10----level--0----------------------------------------------main-(start sequence)---------------                                                 

   //-step-10----level--0-------------------------------------------------------------                                                 
   //            ID: init idle sequence
   //---------------------------------------------------------------------------------                                                 
           10  :                                                     

               // disable automatic mode
               // ---------------------
               "DC".MOD_AUT_ENB := FALSE;

               "DV".LMP_OR := false;     // reset orange lamp on control cabinet 

               #end_of_step[0] := true;                            
               #next_step[0] := 100;


   //-step-100---level--0-------------------------------------------------------------                                                 
   //            ID: wait for manual mode
   //---------------------------------------------------------------------------------                                                 
           100 :                                                     

               IF "APC".AUTOMATIC = FALSE THEN                    // manual mode ?
                   "APC".ACT_TME_PROC := 0;                       // start process time
                   "APC".ACT_TME_STE :=  0;
                   #end_of_step[0] := true;                            
               END_IF;                                    
               #next_step[0] := 200;


   //-step-200---level--0-------------------------------------------------------------                                                 
   //            ID: idle mode
   //---------------------------------------------------------------------------------                                                 
           200 :                                                     
               IF #next_step[0] = #active_step[0] THEN                       
                   "APC".OP_MSG := "OP_MSG".BLANK;

                   // init control loops
                   // ------------------
                   "DC".CTL_DIA_ON       := FALSE;                      // all control loops off
                   "DC".CTL_GRW_RTE_ON   := FALSE;
                   "DC".CTL_PULL_RTE_ON  := FALSE;
                   "DC".CTL_CRUC_ROT_ON  := FALSE;
                   "DC".CTL_MLT_LVL_ON   := FALSE;
                   "DC".CTL_MLT_1_TMP_ON := FALSE;
                   "DC".CTL_MLT_2_TMP_ON := FALSE;
                   "DC".CTL_GAP_ON       := FALSE;

                   "DC".CTL_HTR_1_TMP_ON := FALSE;
                   "DC".CTL_HTR_2_TMP_ON := FALSE;

                   "DC".CTL_PRS_ON       := FALSE;

                   //reset initial temperature and power setpoints
                   //---------------------------------------------
                   "DIS".HTR_1_TMP_SET_PHA_STR   :=  0.0;
                   "DIS".HTR_2_PWR_SET_PHA_STR   :=  0.0;

                   //set miscellaneous variables and flags
                   //-------------------------------------
                   "AC".XT_MENISCUS := 0.0;

                   "FLT".CAM_THR_ADJ_STOPPED  := FALSE;   // reset fault messages
                   "FLT".CAM_THR_ADJ_ABORTED  := FALSE; 
                   "DV".THR_CALC_DISABLED     := TRUE;    //threshold calculation in this step is disabled

                   "DC".V1_OPEN_REQ   := FALSE;           // only EKZ 2700
                   "DC".V1_CLOSE_REQ  := FALSE;

               END_IF;

               #next_step[0] := 200; 

   //---------------------------------------------------------------------------------                                                 
   //---------------------------------------------------------------------------------                                                 

   //-error------level--0---------------------------------------------------(error in level 0)-------------
       ELSE:                                                        
           //error code                                                //do error code
           ;        
   //------------------------------------------------------------------------------------------------------
       END_CASE;


       #start_previous := #start;                                    //save start input for next call 
       #cont_previous := "APC".CONT;                                  //save cont input for next call 
       #resume_previous := "APC".RESUME;                              //save resume input for next call
       #jump_previous := "APC".JUMP;                                  //save jump input for next call
       #single_previous := "APC".SINGLE;                              //save single input for next call
END_FUNCTION_BLOCK

FUNCTION_BLOCK "AM_PD"   // FB196, SCL
{ S7_Optimized_Access := 'FALSE' }
VERSION : 0.0
// --------------------------------------------------------------------------------
//     program     :    AM_PD
//     description :    apc pump down module  
//     name        :    K. Kalkowski
//     date        :    24.08.99
// 
//     revision    :    call AM_SEQUENCE_CTL
//     name        :    D. Bruess
//     date        :    26.10.99
//                     (c)CGS
//     --------------------------------------------------------------------------------
   VAR_INPUT
      start : Bool;   // start sequence, activate step 10 (impulse triggered)
   END_VAR
   VAR
      start_previous : Bool;   // start input value of last call
      cont_previous : Bool;   // cont input value of last call
      resume_previous : Bool;   // resume input value of last call
      jump_previous : Bool;   // jump input value of last call
      single_previous : Bool;   // single input value of last call
      active_step : Array[0..7] of Int;   // active step number for sequence level 0..7
      next_step : Array[0..7] of Int;   // next step number for sequence level 0..7
      hold_step : Array[0..7] of Int;   // step number of step on hold
      end_of_step : Array[0..7] of Bool;   // active step is done flag for sequence 0..7
      EndOfStep : Bool;   // default value for active step is done flag
      cont_enable : Array[0..7] of Bool;   // enable continue function
      ContEnable : Bool;   // default value for enable continue function
      CAL_CYC_FLAG : Bool;   // 10 sec. cycle flag for drive cal
      fdr_ok : Bool;   // true if feeder is in home position
      prg_cyc_cnt : Int;
      cal_cyc_tme_dly : Int;   // actual time of cycle timer
      prs_leak_test_start : Real;   // pressure at start of leak test
   END_VAR
   VAR_TEMP
      dummy_bool : Bool;   // not used bit
   END_VAR
BEGIN


       "APC".STATUS := "APC".PUMP_DOWN;                                // set apc status               

       "AM_SEQUENCE_CTL" (start_p            := #start,               // control sequence
                        start_previous_p   := #start_previous,
                        cont_previous_p    := #cont_previous, 
                        resume_previous_p  := #resume_previous,
                        jump_previous_p    := #jump_previous,
                        single_previous_p  := #single_previous,
                        active_step_p      := #active_step, 
                        next_step_p        := #next_step,
                        hold_step_p        := #hold_step, 
                        end_of_step_p      := #end_of_step, 
                        cont_enable_p      := #cont_enable); 



       CASE #active_step[0] OF    //sequence level_0
   //step--0-----level--0-------------------------------------------------off--(sequence off)--------------
           0    :                                                  
                #next_step[0] := 0;

   //step--1-----level--0-------------------------------------------------hold-(test sequence)-------------
           1   :                                                       
               IF #next_step[0] = #active_step[0] THEN                   //init step     
                   //init code
                   ; 
               END_IF;

               //step code                                             //do step
               ;

   //-step-10----level--0----------------------------------------------main-(start sequence)---------------                                                 

   //-step-10----level--0-------------------------------------------------------------                                                 
   //            PD: init pump down sequence
   //---------------------------------------------------------------------------------                                                 
           10  :                                                     

               // init vacuum system
               // ------------------
               "DC".V3_OP    := FALSE;
               "DC".V4_OP    := FALSE;
               "DC".V5_OP    := FALSE;
               "DC".V6_OP    := FALSE;
               "DC".V8_OP    := FALSE;
               "DC".V11_OP   := FALSE;
               "DC".V11_CL   := TRUE;
               "DC".V12_OP   := FALSE;
               "DC".V13_OP   := FALSE;
               "DC".V20_OP   := FALSE;
               "DC".V21_OP   := FALSE;
               "DC".V22_OP   := FALSE;
               "DC".V24_OP   := FALSE;
               "DC".P1_ON    := TRUE;                        // start main pump
               //check if bypass filter is activated
               //-----------------------------------
               IF (("CNF".ACT_DVC_CNF AND 2#1000_0000_0000_0000_0000_0000_0000_0000) = 2#1000_0000_0000_0000_0000_0000_0000_0000) THEN 
                   "DC".P3_ON    := TRUE;                    // P3 on for pump down of bypass filter
               ELSE
                   "DC".P3_ON    := FALSE;                   // P3 off
               END_IF;
               "DC".V3_2_OP  := FALSE;                       // vacuum valve feeder
               "DC".V3_4_OP  := FALSE;
               "DC".V1_1_REL := FALSE;

               "DC".V1_OPEN_REQ  := TRUE;                  // only EKZ 2700
               "DC".V1_CLOSE_REQ := FALSE;

               "AC".SET_CTL_VALVE_POS        := 100.0;       //open throttle valve
               "AC".SET_GAS_1_FLW            := 0.0;
               "AC".SET_GAS_2_FLW            := 0.0;
               #prg_cyc_cnt                 := 0;

               // init drives
               // -----------
               "DC".XT_LFT_UP := FALSE;                    // stop crystal lift
               "DC".XT_LFT_DN := FALSE;
               "DC".XT_LFT_FST := FALSE;
               "DC".XT_ROT_CW := FALSE;                    // stop crystal rotation
               "DC".XT_ROT_CCW := FALSE;

               "DC".CR_LFT_UP := FALSE;                    // stop crucible lift
               "DC".CR_LFT_DN := FALSE;
               "DC".CR_LFT_FST := FALSE;
               "DC".CR_ROT_CW := FALSE;                    // stop crucible rotation
               "DC".CR_ROT_CCW := FALSE;

               "AC".SET_XT_SPD := 0.0;
               "AC".SET_XT_ROT := 0.0;
               "AC".SET_CR_SPD := 0.0;
               "AC".SET_CR_ROT := 0.0;

               // init drive calibration
               //-----------------------
               "KYA".SET_XT_LFT_OFS  := 0.0;     //reset offset to 0.0
               "KYA".SET_XT_LFT_GN   := 1.0;     //reset gain to 1.0
               "KYA".SET_XT_ROT_OFS  := 0.0;    
               "KYA".SET_XT_ROT_GN   := 1.0;   
               "KYA".SET_CR_LFT_OFS  := 0.0;  
               "KYA".SET_CR_LFT_GN   := 1.0; 
               "KYA".SET_CR_ROT_OFS  := 0.0; 
               "KYA".SET_CR_ROT_GN   := 1.0; 

               // init heater
               // -----------
               "DC".HTR_1_ON := FALSE;                     // heater off
               "DC".HTR_2_ON := FALSE;
               "DC".HTR_3_ON := FALSE;

               "AC".SET_HTR_1_PWR := 0.0;
               "AC".SET_HTR_2_PWR := 0.0;
               "AC".SET_HTR_3_PWR := 0.0;

               //mobile feeder
               //-------------
               "DC".MOB_FDR_MVE_IN_SEQ_ON    :=  FALSE;
               IF ("LT".MOB_FDR_DCK_DONE AND ("DV".FDG_MVE_IN_SEQ_DONE OR NOT "DV".FDG_MVE_OUT_SEQ_DONE)) THEN 
                   "DC".MOB_FDR_MVE_OUT_SEQ_ON   :=  TRUE;
               ELSE
                   "DC".MOB_FDR_MVE_OUT_SEQ_ON   :=  FALSE;
               END_IF;
               "DC".MOB_FDR_VIB_ON           :=  FALSE;
               "FLT".MOB_FDR_NOT_DCK         :=  FALSE;
               "FLT".MOB_FDR_STP_PARA        :=  FALSE;

               // init magnet
               // -----------
               "DC".MAG_ON := FALSE;                       // magnet off

               "AC".SET_MAG_1_CUR := 0.0;
               "AC".SET_MAG_2_CUR := 0.0;

               // init control loops
               // ------------------
               "DC".CTL_DIA_ON := FALSE;                   // all control loops off
               "DC".CTL_GRW_RTE_ON := FALSE;
               "DC".CTL_PULL_RTE_ON := FALSE;
               "DC".CTL_CRUC_ROT_ON := FALSE;
               "DC".CTL_MLT_LVL_ON := FALSE;
               "DC".CTL_MLT_1_TMP_ON := FALSE;
               "DC".CTL_MLT_2_TMP_ON := FALSE;
               "DC".CTL_MLT_DRIFT_ON := FALSE;
               "DC".CTL_GAP_ON       := FALSE;

               "DC".CTL_HTR_1_TMP_ON := FALSE;
               //DC.CTL_HTR_2_TMP_ON := FALSE;

               "DC".SET_HTR_1_TMP_ABS := TRUE;           // disable inc functions
               "DC".SET_HTR_2_PWR_ABS := TRUE;

               "DC".CTL_PRS_ON := FALSE;

               "DC".CTL_SI_FDR_ON := FALSE;
               "DC".CTL_DOP_FDR_ON := FALSE;

               "AC".SET_XT_DIA := 0.0;
               "AC".SET_GRW_RTE := 0.0;
               "AC".SET_AVG_SPD := 0.0;
               "AC".SET_AVG_CRUC_ROT := 0.0;
               "AC".SET_MLT_LVL_LSR := 0.0;
               "AC".SET_MLT_1_TMP := 0.0;
               "AC".SET_MLT_2_TMP := 0.0;
               "AC".SET_HTR_1_TMP := 0.0;
               "AC".SET_HTR_2_TMP := 0.0;

               // init measurement system
               // -----------------------
               "DC".CAM_ISP_ON   :=  FALSE;      //inspection off
               "DC".CAM_INIT     :=  FALSE;
               //DC.CAM_MLT      :=  TRUE;
               //DC.CAM_DIP      :=  FALSE;
               //DC.CAM_DIA      :=  FALSE;
               "DC".CAM_SEL_1    :=  TRUE;
               "DC".CAM_SEL_2    :=  FALSE;

               "KYA".SET_THR_CAL_FACT    := 1.0;           // default value for threshold ratio factor
               "DV".THR_CALC_DISABLED    := TRUE;            

               "DC".LSR_ON := FALSE;                       // laser off
               "DC".MCC_ON := FALSE;                       // melt contact control off
               "DC".MCC_TST_ON := FALSE;

               // init Si feeder system
               // ---------------------
               "DC".SI_FDR_ON := FALSE;                    // feeder off
               "DC".DOP_FDR_ON := FALSE;

               "AC".SET_FDR_SI := 0.0;
               "AC".SET_FDR_DOP := 0.0;

               // init lamp on control cabinet
               // ----------------------------
               "DV".LMP_OR := false;

               // process control flags
               // ---------------------
               "APC".PNBDY := FALSE;
               "APC".BYRST := FALSE;

               //reset dipping alarms
               //--------------------
               "FLT".DI_IMAGE_TO_DARK    := FALSE;   
               "FLT".DI_ISOLATION_FAULT  := FALSE;   
               "FLT".DI_MCC_ERROR_1      := FALSE;  
               "FLT".DI_MCC_ERROR_2      := FALSE;

               //set tare request
               //----------------
               "DV".XT_WGT_CELL_TAR_REQ  :=  TRUE;

               // calculate all setpoints 
               // -----------------------
               "AM_PAR_FNC_PD" (act_x_value := 0.0);

               // enable automatic mode
               // ---------------------
               // DC.MOD_AUT_ENB := TRUE;                // only if gate valve open

               #end_of_step[0] := true;                            
               #next_step[0] := 50;


   //-step-50----level--0-------------------------------------------------------------                                                 
   //            PD: gate valve open ?
   //---------------------------------------------------------------------------------                                                 
           50 :                                                     
               IF #next_step[0] = #active_step[0] THEN
                   "APC".OP_MSG := "OP_MSG".WAIT_FOR_AUTO;                                                  
               END_IF;

               //reset total, process and step time
               //----------------------------------
               "APC".ACT_TME_TOT     := 0;   //total time
               "APC".ACT_TME_PROC    := 0;   //process time
               "APC".ACT_TME_STE     := 0;   //step time

               // calculate all setpoints 
               // -----------------------
               "AM_PAR_FNC_PD" (act_x_value := 0.0);

               // feeder in home position?          
               #fdr_ok := NOT "DV".FDR_IN_POS OR "DV".FDR_TUBE_HOME_POS; 


               IF ("LT".V7_OPEN  AND #fdr_ok)  THEN         // gate valve open ? 
                   // open, enable automatic mode
                   // ---------------------------
                   "DC".MOD_AUT_ENB := TRUE;
                   "FLT".PD_GATE_VALVE_CLOSED := FALSE;
                   "FLT".FDR_NOT_IN_HOME_POS := FALSE;
                   #end_of_step[0] := true;
               ELSE
                   // closed, set alarm
                   // -----------------
                   IF "LT".V7_CLOSE THEN
                       "APC".OP_MSG := "OP_MSG".OPEN_GATE_VALVE;                                                  
                       "FLT".PD_GATE_VALVE_CLOSED := TRUE;
                   ELSE
                       "FLT".PD_GATE_VALVE_CLOSED := FALSE;
                   END_IF;
                   IF NOT #fdr_ok THEN
                       "APC".OP_MSG := "OP_MSG".MOVE_FDR_TO_HOME;
                       "FLT".FDR_NOT_IN_HOME_POS := TRUE;
                   ELSE
                       "FLT".FDR_NOT_IN_HOME_POS := FALSE;
                   END_IF;

                   "DC".MOD_AUT_ENB := FALSE;
               END_IF;                                    

               #next_step[0] := 100;

   //-step-100---level--0-------------------------------------------------------------                                                 
   //            PD: wait for automatic mode
   //---------------------------------------------------------------------------------                                                 
           100 :                                                     
               IF #next_step[0] = #active_step[0] THEN
                   "APC".OP_MSG := "OP_MSG".WAIT_FOR_AUTO;                                                  
               END_IF;

               // calculate all setpoints 
               // -----------------------
               "AM_PAR_FNC_PD" (act_x_value := 0.0);


               IF "APC".AUTOMATIC    THEN                    // automatic mode ?
                   #end_of_step[0] := true;                            
               END_IF;                                    

               #next_step[0] := 120;

   //-step-120---level--0-------------------------------------------------------------                                                 
   //            PD: select pump down with or without purging
   //---------------------------------------------------------------------------------                                                 
           120 :                                                     
               IF #next_step[0] = #active_step[0] THEN
                   "APC".OP_MSG := "OP_MSG".BLANK;                                                  
               END_IF;

               #end_of_step[0] := true;                            

               //check amount of requested cycles
               //--------------------------------
               IF (REAL_TO_INT("PAR_MAIN".PD_AMT_PRG_CYC) > 0)  THEN
                   #next_step[0] := 140;    //do purging
               ELSE
                   #next_step[0] := 200;    //skip purging 
               END_IF;

   //-step-140---level--0-------------------------------------------------------------                                                 
   //            PD: pump down to selected pressure before purging
   //---------------------------------------------------------------------------------                                                 
           140 :                                                     
               IF #next_step[0] = #active_step[0] THEN
                   "APC".OP_MSG      := "OP_MSG".PD_PRG_PRS; 
                   "APC".ACT_TME_STE := 0;
                   "APC".TI[0]       := 0;              

               END_IF;

               // calculate all setpoints 
               // -----------------------
               "AM_PAR_FNC_PD" (act_x_value := 0.0);

               //open vacuum valve to bypass filter
               //----------------------------------
               IF (("CNF".ACT_DVC_CNF AND 2#1000_0000_0000_0000_0000_0000_0000_0000) = 2#1000_0000_0000_0000_0000_0000_0000_0000) THEN 
                   "DC".V3_4_OP  := TRUE;
               ELSE
                   "DC".V3_4_OP  := FALSE;
               END_IF;

               //check if final pressure is reached
               //----------------------------------
               IF "APC".AUTOMATIC THEN                                               //automatic mode is running
                   IF ("AV".ACT_PRS_FCH <= "PAR_MAIN".PD_PRG_STR_PRS)  THEN
                       "AC".SET_CTL_VALVE_POS        := 0.0;     //close throttle valve

                   ELSE
                       "AC".SET_CTL_VALVE_POS        := 100.0;   //open throttle valve

                   END_IF;

                   IF ("AC".SET_CTL_VALVE_POS = 100.0) THEN
                       "APC".TI[0]   :=  0;
                   END_IF;
               ELSE
                   "APC".TI[0]   :=  0;
               END_IF;

               //check end condition
               //-------------------
               IF ("APC".TI[0] >= 3) THEN                //main vacuum valve closed?
                   #end_of_step[0] := true;                            
               END_IF;

               #next_step[0] := 160;   

   //-step-160---level--0-------------------------------------------------------------                                                 
   //            PD: purge Ar to furnace
   //---------------------------------------------------------------------------------                                                 
           160 :                                                     
               IF #next_step[0] = #active_step[0] THEN
                   "APC".OP_MSG  := "OP_MSG".PD_PRG;       
                   "APC".TI[0]   :=  0;                                           
               END_IF;

               // calculate all setpoints 
               // -----------------------
               "AM_PAR_FNC_PD" (act_x_value := 0.0);

